// TwinCAT 3 PLC project AlternateCoolingSystem
// ProgramVersion: 3.1.4024.0
// libraries:
//   Tc2_Standard, * (Beckhoff Automation GmbH)
//   Tc2_System, * (Beckhoff Automation GmbH)
//   Tc3_Module, * (Beckhoff Automation GmbH)
// project tree:
//   DUTs/ E_TankState.TcDUT, ST_Tank.TcDUT
//   / PlcTask.TcTTO (not stored)
//   POUs/ FB_TankController.TcPOU, F_CheckAlarm.TcPOU, F_CoolTank.TcPOU, I_TankController.TcIO, MAIN.TcPOU
// (motion and I/O tree: see PLC project functionblockpractice)
// real-time tasks:
//   TASK PlcTask: cycle T#10ms, priority 20, ADS port 350
//   TASK PlcTask2: cycle T#10ms, priority 22, ADS port 352
//   TASK PlcTask1: cycle T#10ms, priority 21, ADS port 351
//   TASK PlcTask3: cycle T#10ms, priority 23, ADS port 353
//   TASK PlcTask4: cycle T#10ms, priority 24, ADS port 354
//   TASK PlcTask5: cycle T#10ms, priority 25, ADS port 355
//   TASK PlcTask6: cycle T#10ms, priority 26, ADS port 356
//   TASK PlcTask7: cycle T#10ms, priority 27, ADS port 357

// ---- DUTs/E_TankState.TcDUT
{attribute 'qualified_only'}
{attribute 'strict'}
TYPE E_TankState :
(
	Idle := 0,
	Filling := 1,
	Processing := 2,
	Dispensing := 3,
	Cooling := 4,
	Alarm := 5
);
END_TYPE

// ---- DUTs/ST_Tank.TcDUT
TYPE ST_Tank :
STRUCT
	nId : INT;
	fTemperature : REAL;
	fLevel : REAL;
	bAlarm : BOOL;
	eState : E_TankState;
END_STRUCT
END_TYPE

// ---- POUs/I_TankController.TcIO
INTERFACE I_TankController

METHOD ApplyCooling : BOOL
VAR_INPUT
END_VAR
END_METHOD

METHOD CheckSafety : BOOL
VAR_INPUT
END_VAR
END_METHOD

METHOD TransferChemical : BOOL
VAR_INPUT
END_VAR
END_METHOD

END_INTERFACE

// ---- POUs/FB_TankController.TcPOU
FUNCTION_BLOCK FB_TankController IMPLEMENTS I_TankController


VAR_IN_OUT
	stTank : ST_Tank;
END_VAR
VAR
	eState : E_TankState;
END_VAR


IF __ISVALIDREF(stTank) THEN
	eState := stTank.eState;
	CheckSafety();
	CASE eState OF
		E_TankState.Idle:
		
		IF NOT stTank.bAlarm THEN
			stTank.eState := E_TankState.Filling;
		END_IF
		E_TankState.Filling:
		
		IF NOT stTank.bAlarm THEN
			stTank.eState := E_TankState.Filling;
		END_IF
		E_TankState.Processing:
		
		E_TankState.Dispensing:
		
		E_TankState.Cooling:
		
		E_TankState.Alarm:
	END_CASE

	
END_IF

{warning 'add method implementation '}
METHOD ApplyCooling : BOOL
IF stTank.bAlarm THEN
	F_CoolTank(stTank);
END_IF
END_METHOD

{warning 'add method implementation '}
METHOD CheckSafety : BOOL
IF F_CheckAlarm( pTank := ADR(stTank) ) THEN
	stTank.bAlarm := TRUE;
END_IF
END_METHOD

METHOD TransferChemical : BOOL
VAR_INPUT
END_VAR
END_METHOD

END_FUNCTION_BLOCK

// ---- POUs/F_CoolTank.TcPOU
FUNCTION F_CoolTank : BOOL
VAR_INPUT
	rTank : REFERENCE TO ST_Tank;
END_VAR
VAR
	fCoolingSpeed : REAL := 3;
	fRequiredTemperature : REAL := 50;
END_VAR

IF __ISVALIDREF(rTank) THEN
	IF rTank.fTemperature > fRequiredTemperature THEN
		rTank.fTemperature := rTank.fTemperature - fCoolingSpeed;
	ELSE
		rTank.bAlarm := FALSE;
		rTank.fTemperature := rTank.fTemperature + fCoolingSpeed;
	END_IF
END_IF

END_FUNCTION

// ---- POUs/F_CheckAlarm.TcPOU
FUNCTION F_CheckAlarm : BOOL
VAR_INPUT
	pTank : POINTER TO ST_Tank;
END_VAR
VAR
	fLevel : REAL := pTank^.fLevel;
	fTemperature : REAL := pTank^.fTemperature;
	fMaxTemperature : REAL := 80;
	fMaxLevelPercentage : REAL := 90;
END_VAR


IF pTank <> 0 THEN
	IF (fLevel > fMaxLevelPercentage) OR (fTemperature > fMaxTemperature )THEN
		F_CheckAlarm := TRUE;
	END_IF
END_IF

END_FUNCTION

// ---- POUs/MAIN.TcPOU
PROGRAM MAIN
VAR
	stTank1 : ST_Tank := (nId := 101,fTemperature := 45.5, fLevel := 40, bAlarm := FALSE, eState := E_TankState.Idle );
	stTank2 : ST_Tank  := (nId := 102,fTemperature := 72.5, fLevel := 70, bAlarm := FALSE, eState := E_TankState.Idle );
	stTank3 : ST_Tank  := (nId := 103,fTemperature := 60.4, fLevel := 95, bAlarm := FALSE, eState := E_TankState.Idle );
	
	fbController : FB_TankController();
	
	
	bStart : bool;
END_VAR

IF bStart THEN
	fbController(stTank := stTank1);
	fbController(stTank := stTank2);
	fbController(stTank := stTank3);
	bStart := FALSE;
END_IF

END_PROGRAM
